FUNCTION DayOfWeek : STRING

VAR_INPUT
	Day : INT; //Current day of the week
END_VAR

CASE Day OF
	1: DayOfWeek := 'Maandag';
	2: DayOfWeek := 'Dinsdag';
	3: DayOfWeek := 'Woensdag';
	4: DayOfWeek := 'Donderdag';
	5: DayOfWeek := 'Vrijdag';
	6: DayOfWeek := 'Zaterdag';
	7: DayOfWeek := 'Zondag';
END_CASE

END_FUNCTION

(* stored: Version 1.1.0.1, ProductVersion 3.1.4024.12
   POU DayOfWeek: Id {60aa29e9-921d-4c9c-82c3-f087d4d67eb3}, SpecialFunc None *)
